FUNCTION_BLOCK MOMENTARY (* Momentary-contact push button *)
  (* Standard: 61499-1; Classification: HMI; Function: Pushbutton; Type: Momentary *)
  (* Version 0.0, 2007-08-30, JHC, Holobloc Inc *)
  (* Compiler header: package fb.rt.hmi; import java.awt.*; import java.awt.event.*; *)
  (* Compiler classdef: public class MOMENTARY extends IN_EVENT *)
  (* Compiler Java Sun JDK 1.6.0 *)
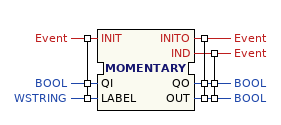
  EVENT_INPUT
    INIT WITH QI, LABEL; (* Service Initialization *)
  END_EVENT
  EVENT_OUTPUT
    INITO WITH QO, OUT; (* Initialization Confirm *)
    IND WITH QO, OUT; (* Event Indication *)
  END_EVENT
  VAR_INPUT
    QI : BOOL := true;
    LABEL : WSTRING; (* Label *)
  END_VAR
  VAR_OUTPUT
    QO : BOOL;
    OUT : BOOL;
  END_VAR
  SERVICE MOMENTARY/Button
    SEQUENCE normal_establishment
      MOMENTARY.INIT+(LABEL) -> Button.setLabel(LABEL) -> MOMENTARY.INITO+();
    END_SEQUENCE
    SEQUENCE normal_termination
      MOMENTARY.INIT-() -> MOMENTARY.INITO-();
    END_SEQUENCE
    SEQUENCE normal_operation
      Button.actionPerformed(QI=1) -> MOMENTARY.IND+(OUT);
    END_SEQUENCE
    SEQUENCE operation_inhibited
      Button.actionPerformed(QI=0);
    END_SEQUENCE
  END_SERVICE
END_FUNCTION_BLOCK
